screen "Home Screen" 1280x800, template "Template_Home"
   Circle "Circle_2" at 219,200 size 21x21
      Appearance <- "DATA_STATUS.LH_SWING_STATUS"
   SymbolLibrary "Symbol Library_1" at 1063,246 size 48x40
      Appearance <- "DATA_STATUS.IDFAN_STATUS"
   SymbolLibrary "Symbol Library_2" at 123,495 size 48x40
      Appearance <- "DATA_STATUS.LHFD_FAN_STATUS"
   SymbolLibrary "Symbol Library_3" at 123,276 size 48x40
      Appearance <- "DATA_STATUS.RHFD_FAN_STATUS"
   SymbolLibrary "Symbol Library_4" at 557,614 size 48x40
      Appearance <- "DATA_STATUS.FP1_STATUS"
   SymbolLibrary "Symbol Library_5" at 640,614 size 48x40
      Appearance <- "DATA_STATUS.FP2_STATUS"
   SymbolLibrary "Symbol Library_6" at 650,562 size 24x33
   SymbolLibrary "Symbol Library_7" at 570,562 size 24x33
   SymbolLibrary "Symbol Library_8" at 570,662 size 24x33
   SymbolLibrary "Symbol Library_9" at 650,662 size 24x33
   SymbolLibrary "Symbol Library_11" at 855,508 size 48x40
      Appearance <- "WORK_BIT.MPA_26"
   TextField "Text Field_8" at 212,700 size 136x22; Text 'from deaerator tank'
   IOField "IO Field_1" at 1037,346 size 97x30; FormatPattern 99.9
      ProcessValue <- "ANALOG_DISPLAY.ID_SPEED"
   TextField "Text Field_10" at 1101,350 size 21x22; Text 'Hz'
   IOField "IO Field_2" at 30,499 size 84x32; FormatPattern 99.9
      ProcessValue <- "ANALOG_DISPLAY.RHFD_SPEED"
   TextField "Text Field_11" at 90,504 size 21x22; Text 'Hz'
   IOField "IO Field_3" at 33,278 size 84x32; FormatPattern 99.9
      ProcessValue <- "ANALOG_DISPLAY.LHFD_SPEED"
   TextField "Text Field_12" at 94,283 size 21x22; Text 'Hz'
   Bar "Bar_1" at 348,299 size 288x126; MinimumValue 0; MaximumValue 100
      ProcessValue <- "ANALOG_DISPLAY.WATER_LEVEL"
   IOField "IO Field_4" at 356,160 size 97x30; FormatPattern 99.9
      ProcessValue <- "ANALOG_DISPLAY.STEAM_PRESSURE"
   TextField "Text Field_13" at 415,164 size 25x22; Text 'bar'
   IOField "IO Field_5" at 686,672 size 71x32; FormatPattern 99.9
      ProcessValue <- "ANALOG_DISPLAY.FP2_SPEED"
   TextField "Text Field_14" at 730,677 size 21x22; Text 'Hz'
   IOField "IO Field_6" at 472,671 size 83x32; FormatPattern 99.9
      ProcessValue <- "ANALOG_DISPLAY.FP1_SPEED"
   TextField "Text Field_15" at 533,676 size 21x22; Text 'Hz'
   IOField "IO Field_7" at 600,444 size 97x32; FormatPattern 99.9
      ProcessValue <- "ANALOG_DISPLAY.RHSTOKER_SPEED"
   IOField "IO Field_8" at 598,249 size 97x30; FormatPattern 99.9
      ProcessValue <- "ANALOG_DISPLAY.LHSTOKER_SPEED"
   TextField "Text Field_16" at 658,253 size 21x22; Text 'Hz'
   TextField "Text Field_17" at 658,449 size 21x22; Text 'Hz'
   Rectangle "Rectangle_5" at 256,196 size 11x23
      Appearance <- "DATA_STATUS.LH_SWING_STATUS"
   TextField "Text Field_18" at 224,203 size 10x14; Text 'M'
   Rectangle "Rectangle_6" at 256,388 size 13x22
      Appearance <- "DATA_STATUS.RH_SWING_STATUS"
   IOField "IO Field_9" at 442,541 size 97x32; FormatPattern 99.9
      ProcessValue <- "ANALOG_DISPLAY.PUMP_PRESSURE"
   TextField "Text Field_20" at 500,546 size 25x22; Text 'bar'
   IOField "IO Field_10" at 386,573 size 153x32; FormatPattern 99.9
      ProcessValue <- "ANALOG_DISPLAY.WATER_FLOWRATE"
   TextField "Text Field_21" at 491,578 size 43x22; Text 'm³/hr'
   IOField "IO Field_11" at 386,605 size 153x32; FormatPattern 999999.9
      ProcessValue <- "ANALOG_DISPLAY.TOTAL_WATER"
   TextField "Text Field_22" at 500,610 size 24x22; Text 'm³'
   IOField "IO Field_12" at 964,111 size 97x32; FormatPattern 99.9
      ProcessValue <- "ANALOG_DISPLAY.O2_LEVEL"
   TextField "Text Field_23" at 1029,116 size 19x22; Text '%'
   IOField "IO Field_13" at 964,143 size 97x32; FormatPattern 99.9
      ProcessValue <- "ANALOG_DISPLAY.CO2_LEVEL"
   TextField "Text Field_24" at 1029,148 size 19x22; Text '%'
   IOField "IO Field_14" at 964,175 size 121x30; FormatPattern 999.9
      ProcessValue <- "ANALOG_DISPLAY.FLUE_GAS_TEMP"
   TextField "Text Field_26" at 925,116 size 22x22; Text 'O²'
   TextField "Text Field_27" at 916,145 size 31x22; Text 'CO²'
   TextField "Text Field_28" at 868,176 size 80x22; Text 'FLUE TEMP'
   TextField "Text Field_29" at 1053,179 size 20x22; Text '°C'
   IOField "IO Field_15" at 173,108 size 153x29; FormatPattern 999999.9
      ProcessValue <- "ANALOG_DISPLAY.LH_TOTAL_COAL"
   TextField "Text Field_30" at 276,112 size 37x22; Text 'Tons'
   IOField "IO Field_16" at 171,299 size 153x29; FormatPattern 999999.9
      ProcessValue <- "ANALOG_DISPLAY.RH_TOTAL_COAL"
   TextField "Text Field_31" at 273,303 size 37x22; Text 'Tons'
   IOField "IO Field_17" at 259,650 size 108x32; FormatPattern 999.9
      ProcessValue <- "ANALOG_DISPLAY.WATER_TEMP"
   IOField "IO Field_18" at 123,422 size 121x30; FormatPattern 999.9
      ProcessValue <- "ANALOG_DISPLAY.RH_BURNBACK_TEMP"
   TextField "Text Field_34" at 199,422 size 10x10; Text 'Text'
   TextField "Text Field_35" at 211,426 size 20x22; Text '°C'
   IOField "IO Field_19" at 121,228 size 121x30; FormatPattern 999.9
      ProcessValue <- "ANALOG_DISPLAY.LH_BURNBACK_TEMP"
   TextField "Text Field_37" at 216,232 size 20x22; Text '°C'
   SymbolLibrary "Symbol Library_14" at 529,166 size 40x33
   GraphicView "Graphics View_23" at 706,181 size 40x22; Picture "3-D Gate valve"
   TextField "Text Field_38" at 368,449 size 83x22; Text 'RH STOKER'
   TextField "Text Field_39" at 358,258 size 81x22; Text 'LH STOKER'
   TextField "Text Field_40" at 1060,381 size 52x22; Text 'ID FAN'
   TextField "Text Field_41" at 37,313 size 76x22; Text 'LH FD FAN'
   TextField "Text Field_42" at 33,535 size 78x22; Text 'RH FD FAN'
   TextField "Text Field_46" at 168,332 size 64x22; Text 'RH COAL'
   TextField "Text Field_48" at 110,399 size 102x22; Text 'RH BURNBACK'
   TextField "Text Field_50" at 914,447 size 91x22; Text 'ASH VALVE 2'
   Circle "Circle_10" at 137,350 size 21x21
      Appearance <- "DATA_STATUS.RHFD_FAN_STATUS"
   TextField "Text Field_3" at 142,353 size 10x14; Text 'M'
   Circle "Circle_8" at 220,392 size 21x21
      Appearance <- "DATA_STATUS.RH_SWING_STATUS"
   TextField "Text Field_19" at 225,395 size 10x14; Text 'M'
   Circle "Circle_11" at 262,450 size 21x21
      Appearance <- "DATA_STATUS.RH_STOKER_STATUS"
   TextField "Text Field_5" at 267,453 size 10x14; Text 'M'
   Circle "Circle_3" at 573,450 size 21x21
      Appearance <- "DATA_STATUS.RH_STOKER_STATUS"
   Circle "Circle_4" at 137,571 size 21x21
      Appearance <- "DATA_STATUS.LHFD_FAN_STATUS"
   TextField "Text Field_1" at 142,574 size 10x14; Text 'M'
   Circle "Circle_7" at 1077,324 size 21x21
      Appearance <- "DATA_STATUS.IDFAN_STATUS"
   TextField "Text Field_7" at 1081,326 size 12x16; Text 'M'
   Circle "Circle_5" at 947,420 size 21x21
      Appearance <- "DATA_STATUS.RAV2_STATUS"
   TextField "Text Field_61" at 951,422 size 12x16; Text 'M'
   Circle "Circle_6" at 702,526 size 21x21
      Appearance <- "DATA_STATUS.RAV1_STATUS"
   TextField "Text Field_2" at 706,528 size 12x16; Text 'M'
   Button "Button_1" at 0,730 size 98x68; TextOff 'Text'; PictureOn "Home_1"; PictureOff "Home_1"
      on Click: ActivateScreen("Home Screen", 0)
   Button "Button_2" at 98,730 size 100x68; TextOn 'Pumps'; TextOff 'Pumps'
      on Click: ActivateScreen("Feed Pump", 0)
   Button "Button_3" at 198,730 size 90x68; TextOn 'Fans'; TextOff 'Fans'
      on Click: ActivateScreen("ID FD Fan", 0)
   Button "Button_4" at 288,730 size 100x68; TextOn 'Stoker'; TextOff 'Stoker'
      on Click: ActivateScreen("Stoker", 0)
   Button "Button_6" at 516,730 size 89x68; TextOff 'Setup'
      on Click: ActivateScreen("Setup", 0)
   Button "Button_11" at 1164,730 size 114x68; TextOff 'Trends'
      on Click: ActivateScreen("Trend Steam", 0)
   Button "Button_5" at 387,730 size 129x68; TextOff 'Coal Handling'
      on Click: ActivateScreen("Coal Handling", 0)
   Button "Button_7" at 604,730 size 210x68; TextOff 'Coal & Blowdown Setup'
      on Click: ActivateScreen("Coal Setup", 0)
   Button "Button_8" at 814,730 size 140x68; TextOff 'Front/Rear Undergrate'
      on Click: ActivateScreen("Front Undergrate Damper", 0)
   Button "Button_20" at 954,730 size 100x68; TextOff 'Alarm Setup'
      on Click: ActivateScreen("Alarm Setup", 0)
   Button "Button_21" at 1054,730 size 110x68; TextOff 'Alarm History'
      on Click: ActivateScreen("Alarm History", 0)
   TextField "Text Field_52" at 675,554 size 91x22; Text 'ASH VALVE 1'
   Circle "Circle_9" at 580,517 size 21x21
      Appearance <- "DATA_STATUS.ASH_CONV_STATUS"
   TextField "Text Field_43" at 584,519 size 12x16; Text 'M'
   TextField "Text Field_44" at 463,516 size 113x22; Text 'ASH CONVEYOR'
   TextField "Text Field_51" at 688,650 size 94x22; Text 'FEED PUMP 2'
   TextField "Text Field_53" at 461,649 size 94x22; Text 'FEED PUMP 1'
   TextField "Text Field_47" at 274,609 size 106x22; Text 'TOTAL WATER'
   TextField "Text Field_54" at 245,578 size 135x22; Text 'WATER FLOWRATE'
   TextField "Text Field_55" at 323,547 size 115x22; Text 'PUMP PRESSURE'
   TextField "Text Field_56" at 84,376 size 128x22; Text 'RH SWING CHUTE'
   TextField "Text Field_45" at 115,203 size 100x22; Text 'LH BURNBACK'
   TextField "Text Field_49" at 89,180 size 126x22; Text 'LH SWING CHUTE'
   TextField "Text Field_57" at 167,145 size 62x22; Text 'LH COAL'
   TextField "Text Field_58" at 358,134 size 124x22; Text 'STEAM PRESSURE'
   TextField "Text field_59" at 646,410 size 13x22; Text '0'
   TextField "Text field_60" at 642,388 size 21x22; Text '20'
   TextField "Text field_62" at 642,363 size 21x22; Text '40'
   TextField "Text field_63" at 642,338 size 21x22; Text '60'
   TextField "Text field_64" at 642,313 size 21x22; Text '80'
   TextField "Text field_65" at 638,288 size 29x22; Text '100'
   GraphicView "Graphic view_2" at 1184,120 size 66x412; Picture "Graphic_4"
   GraphicView "Graphic view_1" at 1178,513 size 80x14; Picture "Graphic_5"
   Button "Button_9" at 914,504 size 99x58; TextOff 'AUTOMATIC BLOWDOWN'
      on Click: function_efd93a16("Automatic Blowdown", 900, 370, -1, -1, 1)
   Circle "Circle_12" at 565,258 size 22x22
      Appearance <- "DATA_STATUS.LH_STOKER_STATUS"
   TextField "Text field_6" at 545,335 size 42x50; Text '%'
   IOField "IO Field_20" at 415,334 size 121x49; FormatPattern 999.9
      ProcessValue <- "ANALOG_DISPLAY.WATER_LEVEL"
   Circle "Circle_1" at 255,258 size 22x22
      Appearance <- "DATA_STATUS.LH_STOKER_STATUS"
   TextField "Text Field_4" at 261,262 size 10x14; Text 'M'
   TextField "Text Field_9" at 338,655 size 20x22; Text '°C'
   Button "Button_10" at 107,226 size 149x36; TextOff 'Text'
      on Click: function_efd93a16("BURN_BACK_OFFSET LH", 249, 122, -1, -1, 1)
   Button "Button_12" at 108,421 size 149x36; TextOff 'Text'
      on Click: function_efd93a16("BURN_BACK_OFFSET RH", 240, 436, -1, -1, 1)

screen "Alarm History" 1280x800, template "Template_All"
   TextField "Text Field_1" at 455,109 size 290x50; Text 'ALARM HISTORY'
   AlarmView "Alarm View_1" at 20,182 size 1244x536; ColumnTextDevice 'PLC'; ColumnTextAckGroup 'GR'; ColumnTextAlarmState 'Status'; ColumnTextAlarmText 'Text'; ColumnTextTime 'Time'; ColumnTextDate 'Date'; ColumnTextNumber 'No.'; AlarmLog "Alarm_History"
   Button "Button_1" at 0,730 size 98x68; TextOff 'Text'; PictureOn "Home_1"; PictureOff "Home_1"
      on Click: ActivateScreen("Home Screen", 0)
   Button "Button_2" at 98,730 size 100x68; TextOn 'Pumps'; TextOff 'Pumps'
      on Click: ActivateScreen("Feed Pump", 0)
   Button "Button_3" at 198,730 size 90x68; TextOn 'Fans'; TextOff 'Fans'
      on Click: ActivateScreen("ID FD Fan", 0)
   Button "Button_4" at 288,730 size 100x68; TextOn 'Stoker'; TextOff 'Stoker'
      on Click: ActivateScreen("Stoker", 0)
   Button "Button_6" at 516,730 size 89x68; TextOff 'Setup'
      on Click: ActivateScreen("Setup", 0)
   Button "Button_11" at 1164,730 size 114x68; TextOff 'Trends'
      on Click: ActivateScreen("Trend Steam", 0)
   Button "Button_18" at 387,730 size 129x68; TextOff 'Coal Handling'
      on Click: ActivateScreen("Coal Handling", 0)
   Button "Button_5" at 604,730 size 210x68; TextOff 'Coal & Blowdown Setup'
      on Click: ActivateScreen("Coal Setup", 0)
   Button "Button_19" at 814,730 size 140x68; TextOff 'Front/Rear Undergrate'
      on Click: ActivateScreen("Front Undergrate Damper", 0)
   Button "Button_20" at 954,730 size 100x68; TextOff 'Alarm Setup'
      on Click: ActivateScreen("Alarm Setup", 0)
   Button "Button_21" at 1054,730 size 110x68; TextOff 'Alarm History'
      on Click: ActivateScreen("Alarm History", 0)

screen "Feed Pump" 1280x800, template "Template_All"
   TextField "Text Field_1" at 515,108 size 221x50; Text 'FEED PUMPS'
   SymbolLibrary "Symbol Library_4" at 235,404 size 80x66
      Appearance <- "DATA_STATUS.FP1_STATUS"
   SymbolLibrary "Symbol Library_5" at 365,404 size 80x66
      Appearance <- "DATA_STATUS.FP2_STATUS"
   SymbolLibrary "Symbol Library_1" at 251,525 size 40x59
   SymbolLibrary "Symbol Library_2" at 387,525 size 40x59
   SymbolLibrary "Symbol Library_3" at 255,297 size 40x59
   SymbolLibrary "Symbol Library_8" at 387,297 size 40x59
   TextField "Text Field_2" at 43,614 size 146x22; Text 'From Deaerator Tank'
   Bar "Bar_1" at 616,253 size 208x373; MinimumValue 0; MaximumValue 100
      ProcessValue <- "ANALOG_DISPLAY.WATER_LEVEL"
   TextField "Text Field_3" at 636,219 size 143x37; Text 'Water Level'
   IOField "IO Field_12" at 632,632 size 172x41; FormatPattern 999.9
      ProcessValue <- "ANALOG_DISPLAY.WATER_LEVEL"
   TextField "Text Field_23" at 754,634 size 28x34; Text '%'
   IOField "IO Field_6" at 89,425 size 112x36; FormatPattern 99.9
      ProcessValue <- "ANALOG_DISPLAY.FP1_SPEED"
   TextField "Text Field_15" at 165,429 size 32x34; Text 'Hz'
   IOField "IO Field_7" at 475,425 size 112x36; FormatPattern 99.9
      ProcessValue <- "ANALOG_DISPLAY.FP2_SPEED"
   TextField "Text Field_16" at 547,429 size 32x34; Text 'Hz'
   Switch "Switch_1" at 910,268 size 240x79; TextOn 'AUTO'; CaptionText 'Switch'; TextOff 'HAND'
      ProcessValue <- "DATA_SWITCH.AUTO_FP"
      Appearance <- "DATA_SWITCH.AUTO_FP"
   Button "Button_8" at 910,349 size 240x79; TextOff 'SPEED UP'
      on Press: function_dd21b452("DATA_PARAMETER.HAND_REFF_FP", 2); function_b14e0dd5("PUMP_SPEED_UP", 0)
      Appearance <- "PUMP_SPEED_UP"
   Button "Button_9" at 910,430 size 240x79; TextOff 'SPEED DOWN'
      on Press: function_b9b71300("DATA_PARAMETER.HAND_REFF_FP", 2); function_b14e0dd5("PUMP_SPEED_DOWN", 0)
      Appearance <- "PUMP_SPEED_DOWN"
   IOField "IO Field_10" at 910,581 size 210x43; FormatPattern 99.9
      ProcessValue <- "ANALOG_DISPLAY.WATER_FLOWRATE"
   TextField "Text Field_21" at 1028,585 size 70x34; Text 'm³/hr'
   IOField "IO Field_11" at 245,668 size 192x39; FormatPattern 999999.9
      ProcessValue <- "ANALOG_DISPLAY.TOTAL_WATER"
   TextField "Text Field_22" at 386,669 size 37x34; Text 'm³'
   IOField "IO Field_9" at 289,206 size 110x38; FormatPattern 99.9
      ProcessValue <- "ANALOG_DISPLAY.PUMP_PRESSURE"
   TextField "Text Field_20" at 355,209 size 40x34; Text 'bar'
   TextField "Text Field_4" at 924,542 size 173x34; Text 'Water Flowrate'
   TextField "Text Field_5" at 253,167 size 194x37; Text 'Pumps Pressure'
   TextField "Text Field_6" at 73,356 size 160x70; Text 'Feed Pump 1 Speed'
   TextField "Text Field_7" at 453,356 size 160x70; Text 'Feed Pump 2 Speed'
   TextField "Text Field_9" at 267,630 size 143x37; Text 'Total Water'
   Button "Button_1" at 0,730 size 98x68; TextOff 'Text'; PictureOn "Home_1"; PictureOff "Home_1"
      on Click: ActivateScreen("Home Screen", 0)
   Button "Button_2" at 98,730 size 100x68; TextOn 'Pumps'; TextOff 'Pumps'
      on Click: ActivateScreen("Feed Pump", 0)
   Button "Button_3" at 198,730 size 90x68; TextOn 'Fans'; TextOff 'Fans'
      on Click: ActivateScreen("ID FD Fan", 0)
   Button "Button_4" at 288,730 size 100x68; TextOn 'Stoker'; TextOff 'Stoker'
      on Click: ActivateScreen("Stoker", 0)
   Button "Button_6" at 516,730 size 89x68; TextOff 'Setup'
      on Click: ActivateScreen("Setup", 0)
   Button "Button_11" at 1164,730 size 114x68; TextOff 'Trends'
      on Click: ActivateScreen("Trend Steam", 0)
   Button "Button_5" at 387,730 size 129x68; TextOff 'Coal Handling'
      on Click: ActivateScreen("Coal Handling", 0)
   Button "Button_7" at 605,730 size 210x68; TextOff 'Coal & Blowdown Setup'
      on Click: ActivateScreen("Coal Setup", 0)
   Button "Button_10" at 814,730 size 140x68; TextOff 'Front/Rear Undergrate'
      on Click: ActivateScreen("Front Undergrate Damper", 0)
   Button "Button_20" at 954,730 size 100x68; TextOff 'Alarm Setup'
      on Click: ActivateScreen("Alarm Setup", 0)
   Button "Button_21" at 1054,730 size 110x68; TextOff 'Alarm History'
      on Click: ActivateScreen("Alarm History", 0)

screen "Trend Steam" 1280x800, template "Template_All"
   Button "Button_1" at 4,735 size 182x64; TextOff 'Pumps'; PictureOff "Home_2"
      on Click: ActivateScreen("Home Screen", 0)
   Button "Button_2" at 550,735 size 182x64; TextOff 'Water Flow Trend'
      on Click: ActivateScreen("Trend Water Flow", 0)
   Button "Button_3" at 4,670 size 182x63; TextOff 'ID Fan Trend'
      on Click: ActivateScreen("Trend ID Fan", 0)
   Button "Button_4" at 732,735 size 182x64; TextOff 'Water Level Trend'
      on Click: ActivateScreen("Trend Water Level", 0)
   Button "Button_5" at 1096,735 size 182x64; TextOff 'Oxygen Level Trend'
      on Click: ActivateScreen("Trend O²", 0)
   Button "Button_6" at 914,735 size 182x64; TextOff 'Flue Temp Trend'
      on Click: ActivateScreen("Trend Flue Gas", 0)
   Button "Button_7" at 914,670 size 182x64; TextOff 'Water Temp Trend'
      on Click: ActivateScreen("Trend Water Temp", 0)
   TextField "Text Field_1" at 455,110 size 440x50; Text 'STEAM PRESSURE TREND'
   TrendView "Trend View_1" at 0,170 size 1280x490
   Button "Button_8" at 368,735 size 182x64; TextOff 'RH Stoker Trend'
      on Click: ActivateScreen("Trend RH Stoker", 0)
   Button "Button_9" at 186,735 size 182x64; TextOff 'LH Stoker Trend'
      on Click: ActivateScreen("Trend LH Stoker", 0)
   Button "Button_10" at 368,670 size 182x64; TextOff 'RH FD Fan Trend'
      on Click: ActivateScreen("Trend RH FD Fan", 0)
   Button "Button_11" at 186,670 size 182x64; TextOff 'LH FD Fan Trend'
      on Click: ActivateScreen("Trend LH FD Fan", 0)
   Button "Button_13" at 1096,670 size 182x64; TextOff 'CO² Level Trend'
      on Click: ActivateScreen("Trend CO²", 0)
   Button "Button_14" at 550,670 size 182x64; TextOff 'Feed Pump Speed Trend'
      on Click: ActivateScreen("Trend Pump Speed", 0)
   Button "Button_15" at 732,670 size 182x64; TextOff 'Pump Press Trend'
      on Click: ActivateScreen("Trend Pump Pressure", 0)

screen "Trend CO²" 1280x800, template "Template_All"
   TextField "Text Field_1" at 496,110 size 318x50; Text 'CO² LEVEL TREND'
   TrendView "Trend View_1" at 0,170 size 1280x490
   Button "Button_13" at 1096,670 size 182x64; TextOff 'Steam Press Trend'
      on Click: ActivateScreen("Trend Steam", 0)
   Button "Button_1" at 4,735 size 182x64; TextOff 'Pumps'; PictureOff "Home_2"
      on Click: ActivateScreen("Home Screen", 0)
   Button "Button_2" at 550,735 size 182x64; TextOff 'Water Flow Trend'
      on Click: ActivateScreen("Trend Water Flow", 0)
   Button "Button_3" at 4,670 size 182x63; TextOff 'ID Fan Trend'
      on Click: ActivateScreen("Trend ID Fan", 0)
   Button "Button_4" at 732,735 size 182x64; TextOff 'Water Level Trend'
      on Click: ActivateScreen("Trend Water Level", 0)
   Button "Button_5" at 1096,735 size 182x64; TextOff 'Oxygen Level Trend'
      on Click: ActivateScreen("Trend O²", 0)
   Button "Button_6" at 914,735 size 182x64; TextOff 'Flue Temp Trend'
      on Click: ActivateScreen("Trend Flue Gas", 0)
   Button "Button_7" at 914,670 size 182x64; TextOff 'Water Temp Trend'
      on Click: ActivateScreen("Trend Water Temp", 0)
   Button "Button_8" at 368,735 size 182x64; TextOff 'RH Stoker Trend'
      on Click: ActivateScreen("Trend RH Stoker", 0)
   Button "Button_9" at 186,735 size 182x64; TextOff 'LH Stoker Trend'
      on Click: ActivateScreen("Trend LH Stoker", 0)
   Button "Button_10" at 368,670 size 182x64; TextOff 'RH FD Fan Trend'
      on Click: ActivateScreen("Trend RH FD Fan", 0)
   Button "Button_11" at 186,670 size 182x64; TextOff 'LH FD Fan Trend'
      on Click: ActivateScreen("Trend LH FD Fan", 0)
   Button "Button_14" at 550,670 size 182x64; TextOff 'Feed Pump Speed Trend'
      on Click: ActivateScreen("Trend Pump Speed", 0)
   Button "Button_15" at 732,670 size 182x64; TextOff 'Pump Press Trend'
      on Click: ActivateScreen("Trend Pump Pressure", 0)

screen "Trend Flue Gas" 1280x800, template "Template_All"
   TextField "Text Field_1" at 481,112 size 405x50; Text 'FLUE GAS TEMP TREND'
   TrendView "Trend View_1" at 0,170 size 1280x490
   Button "Button_6" at 914,735 size 182x64; TextOff 'Steam Press Trend'
      on Click: ActivateScreen("Trend Steam", 0)
   Button "Button_1" at 4,735 size 182x64; TextOff 'Pumps'; PictureOff "Home_2"
      on Click: ActivateScreen("Home Screen", 0)
   Button "Button_2" at 550,735 size 182x64; TextOff 'Water Flow Trend'
      on Click: ActivateScreen("Trend Water Flow", 0)
   Button "Button_3" at 4,670 size 182x63; TextOff 'ID Fan Trend'
      on Click: ActivateScreen("Trend ID Fan", 0)
   Button "Button_4" at 732,735 size 182x64; TextOff 'Water Level Trend'
      on Click: ActivateScreen("Trend Water Level", 0)
   Button "Button_5" at 1096,735 size 182x64; TextOff 'Oxygen Level Trend'
      on Click: ActivateScreen("Trend O²", 0)
   Button "Button_8" at 914,670 size 182x64; TextOff 'Water Temp Trend'
      on Click: ActivateScreen("Trend Water Temp", 0)
   Button "Button_9" at 368,735 size 182x64; TextOff 'RH Stoker Trend'
      on Click: ActivateScreen("Trend RH Stoker", 0)
   Button "Button_10" at 186,735 size 182x64; TextOff 'LH Stoker Trend'
      on Click: ActivateScreen("Trend LH Stoker", 0)
   Button "Button_11" at 368,670 size 182x64; TextOff 'RH FD Fan Trend'
      on Click: ActivateScreen("Trend RH FD Fan", 0)
   Button "Button_12" at 186,670 size 182x64; TextOff 'LH FD Fan Trend'
      on Click: ActivateScreen("Trend LH FD Fan", 0)
   Button "Button_13" at 1096,670 size 182x64; TextOff 'CO² Level Trend'
      on Click: ActivateScreen("Trend CO²", 0)
   Button "Button_14" at 550,670 size 182x64; TextOff 'Feed Pump Speed Trend'
      on Click: ActivateScreen("Trend Pump Speed", 0)
   Button "Button_15" at 732,670 size 182x64; TextOff 'Pump Press Trend'
      on Click: ActivateScreen("Trend Pump Pressure", 0)

screen "Trend ID Fan" 1280x800, template "Template_All"
   TrendView "Trend View_1" at 0,170 size 1280x490
   TextField "Text Field_1" at 482,113 size 376x50; Text 'ID FAN SPEED TREND'
   Button "Button_3" at 4,670 size 182x64; TextOff 'Steam Press Trend'
      on Click: ActivateScreen("Trend Steam", 0)
   Button "Button_1" at 4,735 size 182x64; TextOff 'Pumps'; PictureOff "Home_2"
      on Click: ActivateScreen("Home Screen", 0)
   Button "Button_2" at 550,735 size 182x64; TextOff 'Water Flow Trend'
      on Click: ActivateScreen("Trend Water Flow", 0)
   Button "Button_5" at 732,735 size 182x64; TextOff 'Water Level Trend'
      on Click: ActivateScreen("Trend Water Level", 0)
   Button "Button_6" at 1096,735 size 182x64; TextOff 'Oxygen Level Trend'
      on Click: ActivateScreen("Trend O²", 0)
   Button "Button_7" at 914,735 size 182x64; TextOff 'Flue Temp Trend'
      on Click: ActivateScreen("Trend Flue Gas", 0)
   Button "Button_8" at 914,670 size 182x64; TextOff 'Water Temp Trend'
      on Click: ActivateScreen("Trend Water Temp", 0)
   Button "Button_9" at 368,735 size 182x64; TextOff 'RH Stoker Trend'
      on Click: ActivateScreen("Trend RH Stoker", 0)
   Button "Button_10" at 186,735 size 182x64; TextOff 'LH Stoker Trend'
      on Click: ActivateScreen("Trend LH Stoker", 0)
   Button "Button_11" at 368,670 size 182x64; TextOff 'RH FD Fan Trend'
      on Click: ActivateScreen("Trend RH FD Fan", 0)
   Button "Button_12" at 186,670 size 182x64; TextOff 'LH FD Fan Trend'
      on Click: ActivateScreen("Trend LH FD Fan", 0)
   Button "Button_13" at 1096,670 size 182x64; TextOff 'CO² Level Trend'
      on Click: ActivateScreen("Trend CO²", 0)
   Button "Button_14" at 550,670 size 182x64; TextOff 'Feed Pump Speed Trend'
      on Click: ActivateScreen("Trend Pump Speed", 0)
   Button "Button_15" at 732,670 size 182x64; TextOff 'Pump Press Trend'
      on Click: ActivateScreen("Trend Pump Pressure", 0)

screen "Trend LH Stoker" 1280x800, template "Template_All"
   TrendView "Trend View_1" at 0,170 size 1280x490
   Button "Button_9" at 186,735 size 182x64; TextOff 'Steam Press Trend'
      on Click: ActivateScreen("Trend Steam", 0)
   Button "Button_1" at 4,735 size 182x64; TextOff 'Pumps'; PictureOff "Home_2"
      on Click: ActivateScreen("Home Screen", 0)
   Button "Button_2" at 550,735 size 182x64; TextOff 'Water Flow Trend'
      on Click: ActivateScreen("Trend Water Flow", 0)
   Button "Button_3" at 4,670 size 182x63; TextOff 'ID Fan Trend'
      on Click: ActivateScreen("Trend ID Fan", 0)
   Button "Button_4" at 732,735 size 182x64; TextOff 'Water Level Trend'
      on Click: ActivateScreen("Trend Water Level", 0)
   Button "Button_5" at 1096,735 size 182x64; TextOff 'Oxygen Level Trend'
      on Click: ActivateScreen("Trend O²", 0)
   Button "Button_6" at 914,735 size 182x64; TextOff 'Flue Temp Trend'
      on Click: ActivateScreen("Trend Flue Gas", 0)
   Button "Button_7" at 914,670 size 182x64; TextOff 'Water Temp Trend'
      on Click: ActivateScreen("Trend Water Temp", 0)
   Button "Button_8" at 368,735 size 182x64; TextOff 'RH Stoker Trend'
      on Click: ActivateScreen("Trend RH Stoker", 0)
   Button "Button_11" at 368,670 size 182x64; TextOff 'RH FD Fan Trend'
      on Click: ActivateScreen("Trend RH FD Fan", 0)
   Button "Button_12" at 186,670 size 182x64; TextOff 'LH FD Fan Trend'
      on Click: ActivateScreen("Trend LH FD Fan", 0)
   Button "Button_13" at 1096,670 size 182x64; TextOff 'CO² Level Trend'
      on Click: ActivateScreen("Trend CO²", 0)
   Button "Button_14" at 550,670 size 182x64; TextOff 'Feed Pump Speed Trend'
      on Click: ActivateScreen("Trend Pump Speed", 0)
   Button "Button_15" at 732,670 size 182x64; TextOff 'Pump Press Trend'
      on Click: ActivateScreen("Trend Pump Pressure", 0)
   TextField "Text Field_1" at 465,113 size 450x50; Text 'LH STOKER SPEED TREND'

screen "Trend LH FD Fan" 1280x800, template "Template_All"
   TextField "Text Field_1" at 444,113 size 439x50; Text 'LH FD FAN SPEED TREND'
   TrendView "Trend View_1" at 0,170 size 1280x490
   Button "Button_11" at 186,670 size 182x64; TextOff 'Steam Press Trend'
      on Click: ActivateScreen("Trend Steam", 0)
   Button "Button_1" at 4,735 size 182x64; TextOff 'Pumps'; PictureOff "Home_2"
      on Click: ActivateScreen("Home Screen", 0)
   Button "Button_2" at 550,735 size 182x64; TextOff 'Water Flow Trend'
      on Click: ActivateScreen("Trend Water Flow", 0)
   Button "Button_3" at 4,670 size 182x63; TextOff 'ID Fan Trend'
      on Click: ActivateScreen("Trend ID Fan", 0)
   Button "Button_4" at 732,735 size 182x64; TextOff 'Water Level Trend'
      on Click: ActivateScreen("Trend Water Level", 0)
   Button "Button_5" at 1096,735 size 182x64; TextOff 'Oxygen Level Trend'
      on Click: ActivateScreen("Trend O²", 0)
   Button "Button_6" at 914,735 size 182x64; TextOff 'Flue Temp Trend'
      on Click: ActivateScreen("Trend Flue Gas", 0)
   Button "Button_7" at 914,670 size 182x64; TextOff 'Water Temp Trend'
      on Click: ActivateScreen("Trend Water Temp", 0)
   Button "Button_8" at 368,735 size 182x64; TextOff 'RH Stoker Trend'
      on Click: ActivateScreen("Trend RH Stoker", 0)
   Button "Button_9" at 186,735 size 182x64; TextOff 'LH Stoker Trend'
      on Click: ActivateScreen("Trend LH Stoker", 0)
   Button "Button_10" at 368,670 size 182x64; TextOff 'RH FD Fan Trend'
      on Click: ActivateScreen("Trend RH FD Fan", 0)
   Button "Button_13" at 1096,670 size 182x64; TextOff 'CO² Level Trend'
      on Click: ActivateScreen("Trend CO²", 0)
   Button "Button_14" at 550,670 size 182x64; TextOff 'Feed Pump Speed Trend'
      on Click: ActivateScreen("Trend Pump Speed", 0)
   Button "Button_15" at 732,670 size 182x64; TextOff 'Pump Press Trend'
      on Click: ActivateScreen("Trend Pump Pressure", 0)

screen "Trend O²" 1280x800, template "Template_All"
   TextField "Text Field_1" at 468,111 size 391x50; Text 'OXYGEN LEVEL TREND'
   TrendView "Trend View_1" at 0,170 size 1280x490
   Button "Button_5" at 1096,735 size 182x64; TextOff 'Steam Press Trend'
      on Click: ActivateScreen("Trend Steam", 0)
   Button "Button_1" at 4,735 size 182x64; TextOff 'Pumps'; PictureOff "Home_2"
      on Click: ActivateScreen("Home Screen", 0)
   Button "Button_2" at 550,735 size 182x64; TextOff 'Water Flow Trend'
      on Click: ActivateScreen("Trend Water Flow", 0)
   Button "Button_3" at 4,670 size 182x63; TextOff 'ID Fan Trend'
      on Click: ActivateScreen("Trend ID Fan", 0)
   Button "Button_4" at 732,735 size 182x64; TextOff 'Water Level Trend'
      on Click: ActivateScreen("Trend Water Level", 0)
   Button "Button_7" at 914,735 size 182x64; TextOff 'Flue Temp Trend'
      on Click: ActivateScreen("Trend Flue Gas", 0)
   Button "Button_8" at 914,670 size 182x64; TextOff 'Water Temp Trend'
      on Click: ActivateScreen("Trend Water Temp", 0)
   Button "Button_9" at 368,735 size 182x64; TextOff 'RH Stoker Trend'
      on Click: ActivateScreen("Trend RH Stoker", 0)
   Button "Button_10" at 186,735 size 182x64; TextOff 'LH Stoker Trend'
      on Click: ActivateScreen("Trend LH Stoker", 0)
   Button "Button_11" at 368,670 size 182x64; TextOff 'RH FD Fan Trend'
      on Click: ActivateScreen("Trend RH FD Fan", 0)
   Button "Button_12" at 186,670 size 182x64; TextOff 'LH FD Fan Trend'
      on Click: ActivateScreen("Trend LH FD Fan", 0)
   Button "Button_13" at 1096,670 size 182x64; TextOff 'CO² Level Trend'
      on Click: ActivateScreen("Trend CO²", 0)
   Button "Button_14" at 550,670 size 182x64; TextOff 'Feed Pump Speed Trend'
      on Click: ActivateScreen("Trend Pump Speed", 0)
   Button "Button_15" at 732,670 size 182x64; TextOff 'Pump Press Trend'
      on Click: ActivateScreen("Trend Pump Pressure", 0)

screen "Trend Pump Pressure" 1280x800, template "Template_All"
   TextField "Text Field_1" at 456,112 size 441x50; Text 'PUMPS PRESSURE TREND'
   TrendView "Trend View_1" at 0,170 size 1280x490
   Button "Button_15" at 732,670 size 182x64; TextOff 'Steam Press Trend'
      on Click: ActivateScreen("Trend Steam", 0)
   Button "Button_1" at 4,735 size 182x64; TextOff 'Pumps'; PictureOff "Home_2"
      on Click: ActivateScreen("Home Screen", 0)
   Button "Button_2" at 550,735 size 182x64; TextOff 'Water Flow Trend'
      on Click: ActivateScreen("Trend Water Flow", 0)
   Button "Button_3" at 4,670 size 182x63; TextOff 'ID Fan Trend'
      on Click: ActivateScreen("Trend ID Fan", 0)
   Button "Button_4" at 732,735 size 182x64; TextOff 'Water Level Trend'
      on Click: ActivateScreen("Trend Water Level", 0)
   Button "Button_5" at 1096,735 size 182x64; TextOff 'Oxygen Level Trend'
      on Click: ActivateScreen("Trend O²", 0)
   Button "Button_6" at 914,735 size 182x64; TextOff 'Flue Temp Trend'
      on Click: ActivateScreen("Trend Flue Gas", 0)
   Button "Button_7" at 914,670 size 182x64; TextOff 'Water Temp Trend'
      on Click: ActivateScreen("Trend Water Temp", 0)
   Button "Button_8" at 368,735 size 182x64; TextOff 'RH Stoker Trend'
      on Click: ActivateScreen("Trend RH Stoker", 0)
   Button "Button_9" at 186,735 size 182x64; TextOff 'LH Stoker Trend'
      on Click: ActivateScreen("Trend LH Stoker", 0)
   Button "Button_10" at 368,670 size 182x64; TextOff 'RH FD Fan Trend'
      on Click: ActivateScreen("Trend RH FD Fan", 0)
   Button "Button_11" at 186,670 size 182x64; TextOff 'LH FD Fan Trend'
      on Click: ActivateScreen("Trend LH FD Fan", 0)
   Button "Button_13" at 1096,670 size 182x64; TextOff 'CO² Level Trend'
      on Click: ActivateScreen("Trend CO²", 0)
   Button "Button_14" at 550,670 size 182x64; TextOff 'Feed Pump Speed Trend'
      on Click: ActivateScreen("Trend Pump Speed", 0)

screen "Trend Pump Speed" 1280x800, template "Template_All"
   TrendView "Trend View_1" at 0,170 size 1280x490
   TextField "Text Field_1" at 435,112 size 473x50; Text 'FEED PUMPS SPEED TREND'
   Button "Button_14" at 550,670 size 182x64; TextOff 'Steam Press Trend'
      on Click: ActivateScreen("Trend Steam", 0)
   Button "Button_1" at 4,735 size 182x64; TextOff 'Pumps'; PictureOff "Home_2"
      on Click: ActivateScreen("Home Screen", 0)
   Button "Button_2" at 550,735 size 182x64; TextOff 'Water Flow Trend'
      on Click: ActivateScreen("Trend Water Flow", 0)
   Button "Button_3" at 4,670 size 182x63; TextOff 'ID Fan Trend'
      on Click: ActivateScreen("Trend ID Fan", 0)
   Button "Button_4" at 732,735 size 182x64; TextOff 'Water Level Trend'
      on Click: ActivateScreen("Trend Water Level", 0)
   Button "Button_5" at 1096,735 size 182x64; TextOff 'Oxygen Level Trend'
      on Click: ActivateScreen("Trend O²", 0)
   Button "Button_6" at 914,735 size 182x64; TextOff 'Flue Temp Trend'
      on Click: ActivateScreen("Trend Flue Gas", 0)
   Button "Button_7" at 914,670 size 182x64; TextOff 'Water Temp Trend'
      on Click: ActivateScreen("Trend Water Temp", 0)
   Button "Button_8" at 368,735 size 182x64; TextOff 'RH Stoker Trend'
      on Click: ActivateScreen("Trend RH Stoker", 0)
   Button "Button_9" at 186,735 size 182x64; TextOff 'LH Stoker Trend'
      on Click: ActivateScreen("Trend LH Stoker", 0)
   Button "Button_10" at 368,670 size 182x64; TextOff 'RH FD Fan Trend'
      on Click: ActivateScreen("Trend RH FD Fan", 0)
   Button "Button_11" at 186,670 size 182x64; TextOff 'LH FD Fan Trend'
      on Click: ActivateScreen("Trend LH FD Fan", 0)
   Button "Button_13" at 1096,670 size 182x64; TextOff 'CO² Level Trend'
      on Click: ActivateScreen("Trend CO²", 0)
   Button "Button_15" at 732,670 size 182x64; TextOff 'Pump Press Trend'
      on Click: ActivateScreen("Trend Pump Pressure", 0)

screen "Trend RH Stoker" 1280x800, template "Template_All"
   TextField "Text Field_1" at 465,113 size 455x50; Text 'RH STOKER SPEED TREND'
   TrendView "Trend View_1" at 0,170 size 1280x490
   Button "Button_8" at 368,735 size 182x64; TextOff 'Steam Press Trend'
      on Click: ActivateScreen("Trend Steam", 0)
   Button "Button_1" at 4,735 size 182x64; TextOff 'Pumps'; PictureOff "Home_2"
      on Click: ActivateScreen("Home Screen", 0)
   Button "Button_2" at 550,735 size 182x64; TextOff 'Water Flow Trend'
      on Click: ActivateScreen("Trend Water Flow", 0)
   Button "Button_3" at 4,670 size 182x63; TextOff 'ID Fan Trend'
      on Click: ActivateScreen("Trend ID Fan", 0)
   Button "Button_4" at 732,735 size 182x64; TextOff 'Water Level Trend'
      on Click: ActivateScreen("Trend Water Level", 0)
   Button "Button_5" at 1096,735 size 182x64; TextOff 'Oxygen Level Trend'
      on Click: ActivateScreen("Trend O²", 0)
   Button "Button_6" at 914,735 size 182x64; TextOff 'Flue Temp Trend'
      on Click: ActivateScreen("Trend Flue Gas", 0)
   Button "Button_7" at 914,670 size 182x64; TextOff 'Water Temp Trend'
      on Click: ActivateScreen("Trend Water Temp", 0)
   Button "Button_10" at 186,735 size 182x64; TextOff 'LH Stoker Trend'
      on Click: ActivateScreen("Trend LH Stoker", 0)
   Button "Button_11" at 368,670 size 182x64; TextOff 'RH FD Fan Trend'
      on Click: ActivateScreen("Trend RH FD Fan", 0)
   Button "Button_12" at 186,670 size 182x64; TextOff 'LH FD Fan Trend'
      on Click: ActivateScreen("Trend LH FD Fan", 0)
   Button "Button_13" at 1096,670 size 182x64; TextOff 'CO² Level Trend'
      on Click: ActivateScreen("Trend CO²", 0)
   Button "Button_14" at 550,670 size 182x64; TextOff 'Feed Pump Speed Trend'
      on Click: ActivateScreen("Trend Pump Speed", 0)
   Button "Button_15" at 732,670 size 182x64; TextOff 'Pump Press Trend'
      on Click: ActivateScreen("Trend Pump Pressure", 0)

screen "Trend RH FD Fan" 1280x800, template "Template_All"
   TextField "Text Field_1" at 434,113 size 444x50; Text 'RH FD FAN SPEED TREND'
   TrendView "Trend View_1" at 0,170 size 1280x490
   Button "Button_10" at 368,670 size 182x64; TextOff 'Steam Press Trend'
      on Click: ActivateScreen("Trend Steam", 0)
   Button "Button_1" at 4,735 size 182x64; TextOff 'Pumps'; PictureOff "Home_2"
      on Click: ActivateScreen("Home Screen", 0)
   Button "Button_2" at 550,735 size 182x64; TextOff 'Water Flow Trend'
      on Click: ActivateScreen("Trend Water Flow", 0)
   Button "Button_3" at 4,670 size 182x63; TextOff 'ID Fan Trend'
      on Click: ActivateScreen("Trend ID Fan", 0)
   Button "Button_4" at 732,735 size 182x64; TextOff 'Water Level Trend'
      on Click: ActivateScreen("Trend Water Level", 0)
   Button "Button_5" at 1096,735 size 182x64; TextOff 'Oxygen Level Trend'
      on Click: ActivateScreen("Trend O²", 0)
   Button "Button_6" at 914,735 size 182x64; TextOff 'Flue Temp Trend'
      on Click: ActivateScreen("Trend Flue Gas", 0)
   Button "Button_7" at 914,670 size 182x64; TextOff 'Water Temp Trend'
      on Click: ActivateScreen("Trend Water Temp", 0)
   Button "Button_8" at 368,735 size 182x64; TextOff 'RH Stoker Trend'
      on Click: ActivateScreen("Trend RH Stoker", 0)
   Button "Button_9" at 186,735 size 182x64; TextOff 'LH Stoker Trend'
      on Click: ActivateScreen("Trend LH Stoker", 0)
   Button "Button_12" at 186,670 size 182x64; TextOff 'LH FD Fan Trend'
      on Click: ActivateScreen("Trend LH FD Fan", 0)
   Button "Button_13" at 1096,670 size 182x64; TextOff 'CO² Level Trend'
      on Click: ActivateScreen("Trend CO²", 0)
   Button "Button_14" at 550,670 size 182x64; TextOff 'Feed Pump Speed Trend'
      on Click: ActivateScreen("Trend Pump Speed", 0)
   Button "Button_15" at 732,670 size 182x64; TextOff 'Pump Press Trend'
      on Click: ActivateScreen("Trend Pump Pressure", 0)

screen "Trend Water Flow" 1280x800, template "Template_All"
   TrendView "Trend View_1" at 0,170 size 1280x490
   TextField "Text Field_1" at 494,111 size 370x50; Text 'WATER FLOW TREND'
   Button "Button_2" at 550,735 size 182x64; TextOff 'Steam Press Trend'
      on Click: ActivateScreen("Trend Steam", 0)
   Button "Button_1" at 4,735 size 182x64; TextOff 'Pumps'; PictureOff "Home_2"
      on Click: ActivateScreen("Home Screen", 0)
   Button "Button_4" at 4,670 size 182x63; TextOff 'ID Fan Trend'
      on Click: ActivateScreen("Trend ID Fan", 0)
   Button "Button_5" at 732,735 size 182x64; TextOff 'Water Level Trend'
      on Click: ActivateScreen("Trend Water Level", 0)
   Button "Button_6" at 1096,735 size 182x64; TextOff 'Oxygen Level Trend'
      on Click: ActivateScreen("Trend O²", 0)
   Button "Button_7" at 914,735 size 182x64; TextOff 'Flue Temp Trend'
      on Click: ActivateScreen("Trend Flue Gas", 0)
   Button "Button_8" at 914,670 size 182x64; TextOff 'Water Temp Trend'
      on Click: ActivateScreen("Trend Water Temp", 0)
   Button "Button_9" at 368,735 size 182x64; TextOff 'RH Stoker Trend'
      on Click: ActivateScreen("Trend RH Stoker", 0)
   Button "Button_10" at 186,735 size 182x64; TextOff 'LH Stoker Trend'
      on Click: ActivateScreen("Trend LH Stoker", 0)
   Button "Button_11" at 368,670 size 182x64; TextOff 'RH FD Fan Trend'
      on Click: ActivateScreen("Trend RH FD Fan", 0)
   Button "Button_12" at 186,670 size 182x64; TextOff 'LH FD Fan Trend'
      on Click: ActivateScreen("Trend LH FD Fan", 0)
   Button "Button_13" at 1096,670 size 182x64; TextOff 'CO² Level Trend'
      on Click: ActivateScreen("Trend CO²", 0)
   Button "Button_14" at 550,670 size 182x64; TextOff 'Feed Pump Speed Trend'
      on Click: ActivateScreen("Trend Pump Speed", 0)
   Button "Button_15" at 732,670 size 182x64; TextOff 'Pump Press Trend'
      on Click: ActivateScreen("Trend Pump Pressure", 0)

screen "Trend Water Level" 1280x800, template "Template_All"
   TextField "Text Field_1" at 481,111 size 373x50; Text 'WATER LEVEL TREND'
   TrendView "Trend View_1" at 0,170 size 1280x490
   Button "Button_4" at 732,735 size 182x64; TextOff 'Steam Press Trend'
      on Click: ActivateScreen("Trend Steam", 0)
   Button "Button_1" at 4,735 size 182x64; TextOff 'Pumps'; PictureOff "Home_2"
      on Click: ActivateScreen("Home Screen", 0)
   Button "Button_2" at 550,735 size 182x64; TextOff 'Water Flow Trend'
      on Click: ActivateScreen("Trend Water Flow", 0)
   Button "Button_3" at 4,670 size 182x63; TextOff 'ID Fan Trend'
      on Click: ActivateScreen("Trend ID Fan", 0)
   Button "Button_6" at 1096,735 size 182x64; TextOff 'Oxygen Level Trend'
      on Click: ActivateScreen("Trend O²", 0)
   Button "Button_7" at 914,735 size 182x64; TextOff 'Flue Temp Trend'
      on Click: ActivateScreen("Trend Flue Gas", 0)
   Button "Button_8" at 914,670 size 182x64; TextOff 'Water Temp Trend'
      on Click: ActivateScreen("Trend Water Temp", 0)
   Button "Button_9" at 368,735 size 182x64; TextOff 'RH Stoker Trend'
      on Click: ActivateScreen("Trend RH Stoker", 0)
   Button "Button_10" at 186,735 size 182x64; TextOff 'LH Stoker Trend'
      on Click: ActivateScreen("Trend LH Stoker", 0)
   Button "Button_11" at 368,670 size 182x64; TextOff 'RH FD Fan Trend'
      on Click: ActivateScreen("Trend RH FD Fan", 0)
   Button "Button_12" at 186,670 size 182x64; TextOff 'LH FD Fan Trend'
      on Click: ActivateScreen("Trend LH FD Fan", 0)
   Button "Button_13" at 1096,670 size 182x64; TextOff 'CO² Level Trend'
      on Click: ActivateScreen("Trend CO²", 0)
   Button "Button_14" at 550,670 size 182x64; TextOff 'Feed Pump Speed Trend'
      on Click: ActivateScreen("Trend Pump Speed", 0)
   Button "Button_15" at 732,670 size 182x64; TextOff 'Pump Press Trend'
      on Click: ActivateScreen("Trend Pump Pressure", 0)

screen "Trend Water Temp" 1280x800, template "Template_All"
   TextField "Text Field_1" at 481,113 size 363x50; Text 'WATER TEMP TREND'
   TrendView "Trend View_1" at 0,170 size 1280x490
   Button "Button_7" at 914,670 size 182x64; TextOff 'Steam Press Trend'
      on Click: ActivateScreen("Trend Steam", 0)
   Button "Button_1" at 4,735 size 182x64; TextOff 'Pumps'; PictureOff "Home_2"
      on Click: ActivateScreen("Home Screen", 0)
   Button "Button_2" at 550,735 size 182x64; TextOff 'Water Flow Trend'
      on Click: ActivateScreen("Trend Water Flow", 0)
   Button "Button_3" at 4,670 size 182x63; TextOff 'ID Fan Trend'
      on Click: ActivateScreen("Trend ID Fan", 0)
   Button "Button_4" at 732,735 size 182x64; TextOff 'Water Level Trend'
      on Click: ActivateScreen("Trend Water Level", 0)
   Button "Button_5" at 1096,735 size 182x64; TextOff 'Oxygen Level Trend'
      on Click: ActivateScreen("Trend O²", 0)
   Button "Button_6" at 914,735 size 182x64; TextOff 'Flue Temp Trend'
      on Click: ActivateScreen("Trend Flue Gas", 0)
   Button "Button_9" at 368,735 size 182x64; TextOff 'RH Stoker Trend'
      on Click: ActivateScreen("Trend RH Stoker", 0)
   Button "Button_10" at 186,735 size 182x64; TextOff 'LH Stoker Trend'
      on Click: ActivateScreen("Trend LH Stoker", 0)
   Button "Button_11" at 368,670 size 182x64; TextOff 'RH FD Fan Trend'
      on Click: ActivateScreen("Trend RH FD Fan", 0)
   Button "Button_12" at 186,670 size 182x64; TextOff 'LH FD Fan Trend'
      on Click: ActivateScreen("Trend LH FD Fan", 0)
   Button "Button_13" at 1096,670 size 182x64; TextOff 'CO² Level Trend'
      on Click: ActivateScreen("Trend CO²", 0)
   Button "Button_14" at 550,670 size 182x64; TextOff 'Feed Pump Speed Trend'
      on Click: ActivateScreen("Trend Pump Speed", 0)
   Button "Button_15" at 732,670 size 182x64; TextOff 'Pump Press Trend'
      on Click: ActivateScreen("Trend Pump Pressure", 0)

screen "Trend PID FD Fan" 1280x800, template "Template_All"
   TrendView "Trend View_1" at 50,174 size 1186x542
   TextField "Text field_1" at 541,111 size 204x50; Text 'PID FD FAN'
   Button "Button_1" at 0,730 size 98x68; TextOff 'Text'; PictureOn "Home_1"; PictureOff "Home_1"
      on Click: ActivateScreen("Home Screen", 0)
   Button "Button_2" at 98,730 size 100x68; TextOn 'Pumps'; TextOff 'Pumps'
      on Click: ActivateScreen("Feed Pump", 0)
   Button "Button_3" at 198,730 size 90x68; TextOn 'Fans'; TextOff 'Fans'
      on Click: ActivateScreen("ID FD Fan", 0)
   Button "Button_4" at 288,730 size 100x68; TextOn 'Stoker'; TextOff 'Stoker'
      on Click: ActivateScreen("Stoker", 0)
   Button "Button_6" at 516,730 size 89x68; TextOff 'Setup'
      on Click: ActivateScreen("Setup", 0)
   Button "Button_11" at 1164,730 size 114x68; TextOff 'Trends'
      on Click: ActivateScreen("Trend Steam", 0)
   Button "Button_5" at 387,730 size 129x68; TextOff 'Coal Handling'
      on Click: ActivateScreen("Coal Handling", 0)
   Button "Button_7" at 604,730 size 210x68; TextOff 'Coal & Blowdown Setup'
      on Click: ActivateScreen("Coal Setup", 0)
   Button "Button_8" at 814,730 size 140x68; TextOff 'Front/Rear Undergrate'
      on Click: ActivateScreen("Front Undergrate Damper", 0)
   Button "Button_20" at 954,730 size 100x68; TextOff 'Alarm Setup'
      on Click: ActivateScreen("Alarm Setup", 0)
   Button "Button_21" at 1054,730 size 110x68; TextOff 'Alarm History'
      on Click: ActivateScreen("Alarm History", 0)

screen "Trend PID Pump" 1280x800, template "Template_All"
   TrendView "Trend View_1" at 44,174 size 1186x542
   TextField "Text field_1" at 561,113 size 174x50; Text 'PID PUMP'
   Button "Button_1" at 0,730 size 98x68; TextOff 'Text'; PictureOn "Home_1"; PictureOff "Home_1"
      on Click: ActivateScreen("Home Screen", 0)
   Button "Button_2" at 98,730 size 100x68; TextOn 'Pumps'; TextOff 'Pumps'
      on Click: ActivateScreen("Feed Pump", 0)
   Button "Button_3" at 198,730 size 90x68; TextOn 'Fans'; TextOff 'Fans'
      on Click: ActivateScreen("ID FD Fan", 0)
   Button "Button_4" at 288,730 size 100x68; TextOn 'Stoker'; TextOff 'Stoker'
      on Click: ActivateScreen("Stoker", 0)
   Button "Button_6" at 516,730 size 89x68; TextOff 'Setup'
      on Click: ActivateScreen("Setup", 0)
   Button "Button_11" at 1164,730 size 114x68; TextOff 'Trends'
      on Click: ActivateScreen("Trend Steam", 0)
   Button "Button_5" at 387,730 size 129x68; TextOff 'Coal Handling'
      on Click: ActivateScreen("Coal Handling", 0)
   Button "Button_7" at 604,730 size 210x68; TextOff 'Coal & Blowdown Setup'
      on Click: ActivateScreen("Coal Setup", 0)
   Button "Button_8" at 814,730 size 140x68; TextOff 'Front/Rear Undergrate'
      on Click: ActivateScreen("Front Undergrate Damper", 0)
   Button "Button_20" at 954,730 size 100x68; TextOff 'Alarm Setup'
      on Click: ActivateScreen("Alarm Setup", 0)
   Button "Button_21" at 1054,730 size 110x68; TextOff 'Alarm History'
      on Click: ActivateScreen("Alarm History", 0)

screen "Trend PID Stoker" 1280x800, template "Template_All"
   TrendView "Trend View_1" at 44,174 size 1186x542
   TextField "Text field_1" at 544,111 size 215x50; Text 'PID STOKER'
   Button "Button_1" at 0,730 size 98x68; TextOff 'Text'; PictureOn "Home_1"; PictureOff "Home_1"
      on Click: ActivateScreen("Home Screen", 0)
   Button "Button_2" at 98,730 size 100x68; TextOn 'Pumps'; TextOff 'Pumps'
      on Click: ActivateScreen("Feed Pump", 0)
   Button "Button_3" at 198,730 size 90x68; TextOn 'Fans'; TextOff 'Fans'
      on Click: ActivateScreen("ID FD Fan", 0)
   Button "Button_4" at 288,730 size 100x68; TextOn 'Stoker'; TextOff 'Stoker'
      on Click: ActivateScreen("Stoker", 0)
   Button "Button_6" at 516,730 size 89x68; TextOff 'Setup'
      on Click: ActivateScreen("Setup", 0)
   Button "Button_11" at 1164,730 size 114x68; TextOff 'Trends'
      on Click: ActivateScreen("Trend Steam", 0)
   Button "Button_5" at 387,730 size 129x68; TextOff 'Coal Handling'
      on Click: ActivateScreen("Coal Handling", 0)
   Button "Button_7" at 604,730 size 210x68; TextOff 'Coal & Blowdown Setup'
      on Click: ActivateScreen("Coal Setup", 0)
   Button "Button_8" at 814,730 size 140x68; TextOff 'Front/Rear Undergrate'
      on Click: ActivateScreen("Front Undergrate Damper", 0)
   Button "Button_20" at 954,730 size 100x68; TextOff 'Alarm Setup'
      on Click: ActivateScreen("Alarm Setup", 0)
   Button "Button_21" at 1054,730 size 110x68; TextOff 'Alarm History'
      on Click: ActivateScreen("Alarm History", 0)

Template "Template_All" 1280x800
   GraphicView "Template_Graphic view_2" at 316,3 size 194x105; Picture "mXoqcDlI_400x400"
   TextField "Template_Text field_1" at 826,19 size 97x81; Text 'bar'
   IOField "Template_I/O field_3" at 525,2 size 262x99; FormatPattern 99.9
      ProcessValue <- "ANALOG_DISPLAY.STEAM_PRESSURE"
   GraphicView "Template_Graphic view_1" at 10,6 size 125x97; Picture "euroasiatic_jaya"
   GraphicView "Template_Graphic view_3" at 139,7 size 172x96; Picture "ACTOM"
   DateTimeField "Template_Date/time field_1" at 1080,8 size 155x40
   DateTimeField "Template_Date/time field_2" at 1080,63 size 169x40
   Button "Template_Button_2" at 1058,2 size 220x52; TextOff 'Text'
      on Click: function_efd93a16("Change Date Time", 540, 220, -1, -1, 1)
   Button "Template_Button_1" at 1058,57 size 220x52; TextOff 'Text'
      on Click: function_efd93a16("Change Date Time", 540, 220, -1, -1, 1)
   Button "Template_Button_3" at 10,6 size 125x97; TextOff 'Text'
      on Click: StopRuntime(0)

Template "Template_Home" 1280x800
   GraphicView "Template_Graphic view_2" at 316,3 size 194x105; Picture "mXoqcDlI_400x400"
   GraphicView "Template_Graphic view_1" at 10,6 size 125x97; Picture "euroasiatic_jaya"
   GraphicView "Template_Graphic view_3" at 139,7 size 172x96; Picture "ACTOM"
   TextField "Template_Text field_1" at 826,19 size 97x81; Text 'bar'
   IOField "Template_I/O field_3" at 525,2 size 262x99; FormatPattern 99.9
      ProcessValue <- "ANALOG_DISPLAY.STEAM_PRESSURE"
   DateTimeField "Template_Date/time field_1" at 1082,7 size 155x40
   Button "Template_Button_2" at 1058,2 size 220x52; TextOff 'Text'
      on Click: function_efd93a16("Change Date Time", 540, 220, -1, -1, 1)
   DateTimeField "Template_Date/time field_2" at 1082,62 size 169x40
   Button "Template_Button_1" at 1058,57 size 220x52; TextOff 'Text'
      on Click: function_efd93a16("Change Date Time", 540, 220, -1, -1, 1)
   Button "Template_Button_3" at 10,6 size 125x97; TextOff 'Text'
      on Click: StopRuntime(0)

PopupScreen "Automatic Blowdown" 240x240
   Button "Button_1" at 201,9 size 34x26; TextOff 'X'
      on Click: ActivateScreen("Home Screen", 0)
   TextField "Text field_1" at 25,11 size 178x20; Text 'AUTOMATIC BLOWDOWN'
   TextField "Text field_2" at 12,122 size 73x22; Text 'OFF TIME'
   TextField "Text field_3" at 10,149 size 78x22; Text 'OFF PULSE'
   TextField "Text field_14" at 13,175 size 72x22; Text 'ON PULSE'
   TextField "Text field_15" at 16,202 size 65x22; Text 'PERIODE'
   TextField "Text field_16" at 171,120 size 28x22; Text 'min'
   TextField "Text field_17" at 171,147 size 27x22; Text 'sec'
   TextField "Text field_18" at 171,173 size 27x22; Text 'sec'
   TextField "Text field_19" at 165,203 size 40x22; Text 'times'
   Switch "Switch_3" at 75,78 size 89x32; TextOn 'ON'; CaptionText 'Switch'; TextOff 'OFF'
      ProcessValue <- "PB_BLOWDOWN"
      Appearance <- "PB_BLOWDOWN"
   IOField "I/O field_1" at 92,120 size 53x26; FormatPattern 999
      ProcessValue <- "DATA_PARAMETER.OFF_TIME_BLOWDOWN"
   IOField "I/O field_2" at 92,147 size 53x26; FormatPattern 999
      ProcessValue <- "DATA_PARAMETER.OFF_PULSE_BLOWDOWN"
   IOField "I/O field_3" at 92,174 size 53x26; FormatPattern 999
      ProcessValue <- "DATA_PARAMETER.ON_PULSE_BLOWDOWN"
   IOField "I/O field_4" at 92,201 size 53x26; FormatPattern 999
      ProcessValue <- "DATA_PARAMETER.PERIODE"
   Switch "Switch_1" at 75,44 size 89x32; TextOn 'AUTO'; CaptionText 'Switch'; TextOff 'HAND'
      ProcessValue <- "Hand/Auto_Blowdown"
      Appearance <- "Hand/Auto_Blowdown"

PopupScreen "Change Date Time" 402x252
   TextField "Text field_1" at 29,16 size 285x25; Text 'Change system date and time'
   TextField "Text field_2" at 5,81 size 78x25; Text 'Actual :'
   TextField "Text field_3" at 5,142 size 145x25; Text 'Set date time :'
   Button "Button_1" at 344,10 size 47x36; TextOff 'X'
      on Click: function_efd93a16("Change Date Time", 0, 0, -1, -1, 1)
   Button "Button_2" at 12,195 size 374x44; TextOff 'Change'
      on Press: function_b14e0dd5("Set_DTL", 0)
      Appearance <- "Set_DTL"
   IOField "I/O field_1" at 138,136 size 248x38; FormatPattern 9999999999999999999999999999999999999999
      ProcessValue <- "Set_Date_Time"
   IOField "I/O field_2" at 138,75 size 248x38; FormatPattern 9999999999999999999999999999999999999999
      ProcessValue <- "Date_Time_Actual"

PopupScreen "BURN_BACK_OFFSET LH" 240x100
   TextField "Text field_1" at 7,57 size 88x25; Text 'OFFSET :'
   IOField "I/O field_1" at 96,53 size 96x32; FormatPattern 999.9
      ProcessValue <- "LH_BURN_BACK_OFFSET"
   TextField "Text field_2" at 17,13 size 153x25; Text 'LH BURN BACK'
   Button "Button_1" at 183,9 size 46x36; TextOff 'X'
      on Click: function_efd93a16("BURN_BACK_OFFSET LH", 0, 0, -1, -1, 1)

PopupScreen "BURN_BACK_OFFSET RH" 240x100
   TextField "Text field_1" at 7,57 size 88x25; Text 'OFFSET :'
   IOField "I/O field_1" at 96,53 size 96x32; FormatPattern 999.9
      ProcessValue <- "RH_BURN_BACK_OFFSET"
   TextField "Text field_2" at 17,13 size 155x25; Text 'RH BURN BACK'
   Button "Button_1" at 183,9 size 46x36; TextOff 'X'
      on Click: function_efd93a16("BURN_BACK_OFFSET RH", 0, 0, -1, -1, 1)

screen "AI Min Max Setting" 1280x800, template "Template_All"
   TextField "Text field_3" at 401,110 size 533x50; Text 'ANALOG MIN MAX PARAMETER'
   TextField "Text field_2" at 11,273 size 120x25; Text 'Scalling Min'
   TextField "Text field_4" at 11,307 size 124x25; Text 'Scalling Max'
   TextField "Text field_5" at 141,181 size 94x46; Text 'Pressure Steam'
   IOField "I/O field_1" at 141,269 size 96x32; FormatPattern 999999.9
      ProcessValue <- "DB_Scalling_Pressurre_Steam_Min"
   IOField "I/O field_2" at 141,303 size 96x32; FormatPattern 999999.9
      ProcessValue <- "DB_Scalling_Pressure_Steam_Max"
   TextField "Text field_1" at 281,181 size 88x46; Text 'Pressure Pump'
   IOField "I/O field_3" at 285,269 size 96x32; FormatPattern 999999.9
      ProcessValue <- "DB_Scalling_Pressure_Pump_Min"
   IOField "I/O field_4" at 285,303 size 96x32; FormatPattern 999999.9
      ProcessValue <- "DB_Scalling_Pressure_Pump_Max"
   TextField "Text field_6" at 427,181 size 88x46; Text 'Water Flowrate'
   IOField "I/O field_5" at 429,269 size 96x32; FormatPattern 999999.9
      ProcessValue <- "DB_Scalling_Water_Flowrate_Min"
   IOField "I/O field_6" at 429,303 size 96x32; FormatPattern 999999.9
      ProcessValue <- "DB_Scalling_Water_Flowrate_Max"
   TextField "Text field_7" at 573,181 size 76x46; Text 'Feed Pump 1'
   IOField "I/O field_7" at 573,269 size 96x32; FormatPattern 999999.9
      ProcessValue <- "DB_Scalling_Feed_Pump_1_Min"
   IOField "I/O field_8" at 573,303 size 96x32; FormatPattern 999999.9
      ProcessValue <- "DB_Scalling_Feed_Pump_1_Max"
   TextField "Text field_8" at 717,181 size 76x46; Text 'Feed Pump 2'
   IOField "I/O field_9" at 717,269 size 96x32; FormatPattern 999999.9
      ProcessValue <- "DB_Scalling_Feed_Pump_2_Min"
   IOField "I/O field_10" at 717,303 size 96x32; FormatPattern 999999.9
      ProcessValue <- "DB_Scalling_Feed_Pump_2_Max"
   TextField "Text field_9" at 861,181 size 39x46; Text 'ID Fan'
   IOField "I/O field_11" at 861,269 size 96x32; FormatPattern 999999.9
      ProcessValue <- "DB_Scalling_ID_Fan_Min"
   IOField "I/O field_12" at 861,303 size 96x32; FormatPattern 999999.9
      ProcessValue <- "DB_Scalling_ID_Fan_Max"
   TextField "Text field_10" at 1005,181 size 62x46; Text 'LH FD Fan'
   IOField "I/O field_13" at 1005,269 size 96x32; FormatPattern 999999.9
      ProcessValue <- "DB_Scalling_LH_FD_Fan_Min"
   IOField "I/O field_14" at 1005,303 size 96x32; FormatPattern 999999.9
      ProcessValue <- "DB_Scalling_LH_FD_Fan_Max"
   TextField "Text field_11" at 1150,181 size 64x46; Text 'RH FD Fan'
   IOField "I/O field_15" at 1150,269 size 96x32; FormatPattern 999999.9
      ProcessValue <- "DB_Scalling_RH_FD_Fan_Min"
   IOField "I/O field_16" at 1150,303 size 96x32; FormatPattern 999999.9
      ProcessValue <- "DB_Scalling_RH_FD_Fan_Max"
   TextField "Text field_12" at 141,358 size 67x46; Text 'LH Stoker'
   IOField "I/O field_17" at 141,446 size 96x32; FormatPattern 999999.9
      ProcessValue <- "DB_Scalling_LH_Stoker_Min"
   IOField "I/O field_18" at 141,480 size 96x32; FormatPattern 999999.9
      ProcessValue <- "DB_Scalling_LH_Stoker_Max"
   TextField "Text field_13" at 285,358 size 67x46; Text 'RH Stoker'
   IOField "I/O field_19" at 285,446 size 96x32; FormatPattern 999999.9
      ProcessValue <- "DB_Scalling_RH_Stoker_Min"
   IOField "I/O field_20" at 285,480 size 96x32; FormatPattern 999999.9
      ProcessValue <- "DB_Scalling_RH_Stoker_Max"
   TextField "Text field_14" at 429,358 size 61x46; Text 'NRGT Water'
   IOField "I/O field_21" at 429,446 size 96x32; FormatPattern 999999.9
      ProcessValue <- "DB_Scalling_NRGT(Water_Level)_Min"
   IOField "I/O field_22" at 429,480 size 96x32; FormatPattern 999999.9
      ProcessValue <- "DB_Scalling_NRGT(Water_Level)_Max"
   TextField "Text field_15" at 573,358 size 60x46; Text 'O2 Probe'
   IOField "I/O field_23" at 573,446 size 96x32; FormatPattern 999999.9
      ProcessValue <- "DB_Scalling_O2_Probe_Min"
   IOField "I/O field_24" at 573,480 size 96x32; FormatPattern 999999.9
      ProcessValue <- "DB_Scalling_O2_Probe_Max"
   TextField "Text field_16" at 717,358 size 62x46; Text 'Water Temp'
   IOField "I/O field_25" at 717,446 size 96x32; FormatPattern 999999.9
      ProcessValue <- "DB_Scalling_Water_Temp_Min"
   IOField "I/O field_26" at 717,480 size 96x32; FormatPattern 999999.9
      ProcessValue <- "DB_Scalling_Water_Temp_Max"
   TextField "Text field_17" at 861,358 size 56x46; Text 'Flue Temp'
   IOField "I/O field_27" at 861,446 size 96x32; FormatPattern 999999.9
      ProcessValue <- "DB_Scalling_Flue_Min"
   IOField "I/O field_28" at 861,480 size 96x32; FormatPattern 999999.9
      ProcessValue <- "DB_Scalling_Flue_Max"
   TextField "Text field_18" at 1005,358 size 76x46; Text 'LH Thermo'
   IOField "I/O field_29" at 1005,446 size 96x32; FormatPattern 999999.9
      ProcessValue <- "DB_Scalling_LH_Thermocouple_Min"
   IOField "I/O field_30" at 1005,480 size 96x32; FormatPattern 999999.9
      ProcessValue <- "DB_Scalling_LH_Thermocouple_Max"
   TextField "Text field_19" at 1150,358 size 76x46; Text 'RH Thermo'
   IOField "I/O field_31" at 1150,446 size 96x32; FormatPattern 999999.9
      ProcessValue <- "DB_Scalling_RH_Thermocouple_Min"
   IOField "I/O field_32" at 1150,480 size 96x32; FormatPattern 999999.9
      ProcessValue <- "DB_Scalling_RH_Thermocouple_Max"
   TextField "Text field_20" at 141,535 size 112x46; Text 'LH Front Undergrate'
   IOField "I/O field_33" at 141,622 size 96x32; FormatPattern 999999.9
      ProcessValue <- "DB_Scalling_LH_Front_Undergrate_Min"
   IOField "I/O field_34" at 141,656 size 96x32; FormatPattern 999999.9
      ProcessValue <- "DB_Scalling_LH_Front_Undergrate_Max"
   TextField "Text field_21" at 285,535 size 112x46; Text 'RH Front Undergrate'
   IOField "I/O field_35" at 285,622 size 96x32; FormatPattern 999999.9
      ProcessValue <- "DB_Scalling_RH_Front_Undergrate_Min"
   IOField "I/O field_36" at 285,656 size 96x32; FormatPattern 999999.9
      ProcessValue <- "DB_Scalling_RH_Front_Undergrate_Max"
   TextField "Text field_22" at 427,535 size 112x46; Text 'LH Rear Undergrate'
   IOField "I/O field_37" at 429,622 size 96x32; FormatPattern 999999.9
      ProcessValue <- "DB_Scalling_LH_Rear_Undergrate_Min"
   IOField "I/O field_38" at 429,656 size 96x32; FormatPattern 999999.9
      ProcessValue <- "DB_Scalling_LH_Rear_Undergrate_Max"
   TextField "Text field_23" at 573,535 size 112x46; Text 'RH Rear Undergrate'
   IOField "I/O field_39" at 573,622 size 96x32; FormatPattern 999999.9
      ProcessValue <- "DB_Scalling_RH_Rear_Undergrate_Min"
   IOField "I/O field_40" at 573,656 size 96x32; FormatPattern 999999.9
      ProcessValue <- "DB_Scalling_RH_Rear_Undergrate_Max"
   TextField "Text field_25" at 11,239 size 123x25; Text 'Actual Value'
   IOField "I/O field_41" at 141,235 size 96x32; FormatPattern 999999.9
      ProcessValue <- "ANALOG_DISPLAY.STEAM_PRESSURE"
   IOField "I/O field_42" at 285,235 size 96x32; FormatPattern 999999.9
      ProcessValue <- "ANALOG_DISPLAY.PUMP_PRESSURE"
   IOField "I/O field_43" at 429,235 size 96x32; FormatPattern 999999.9
      ProcessValue <- "ANALOG_DISPLAY.WATER_FLOWRATE"
   IOField "I/O field_44" at 573,235 size 96x32; FormatPattern 999999.9
      ProcessValue <- "ANALOG_DISPLAY.FP1_SPEED"
   IOField "I/O field_45" at 717,235 size 96x32; FormatPattern 999999.9
      ProcessValue <- "ANALOG_DISPLAY.FP2_SPEED"
   IOField "I/O field_46" at 861,235 size 96x32; FormatPattern 999999.9
      ProcessValue <- "ANALOG_DISPLAY.ID_SPEED"
   IOField "I/O field_47" at 1005,235 size 96x32; FormatPattern 999999.9
      ProcessValue <- "ANALOG_DISPLAY.LHFD_SPEED"
   IOField "I/O field_48" at 1150,235 size 96x32; FormatPattern 999999.9
      ProcessValue <- "ANALOG_DISPLAY.RHFD_SPEED"
   TextField "Text field_26" at 11,450 size 120x25; Text 'Scalling Min'
   TextField "Text field_27" at 11,484 size 124x25; Text 'Scalling Max'
   TextField "Text field_29" at 11,416 size 123x25; Text 'Actual Value'
   IOField "I/O field_49" at 141,412 size 96x32; FormatPattern 999999.9
      ProcessValue <- "ANALOG_DISPLAY.LHSTOKER_SPEED"
   IOField "I/O field_50" at 285,412 size 96x32; FormatPattern 999999.9
      ProcessValue <- "ANALOG_DISPLAY.RHSTOKER_SPEED"
   IOField "I/O field_51" at 429,412 size 96x32; FormatPattern 999999.9
      ProcessValue <- "ANALOG_DISPLAY.WATER_LEVEL"
   IOField "I/O field_52" at 573,412 size 96x32; FormatPattern 999999.9
      ProcessValue <- "ANALOG_DISPLAY.O2_LEVEL"
   IOField "I/O field_53" at 717,412 size 96x32; FormatPattern 999999.9
      ProcessValue <- "ANALOG_DISPLAY.WATER_TEMP"
   IOField "I/O field_54" at 861,412 size 96x32; FormatPattern 999999.9
      ProcessValue <- "ANALOG_DISPLAY.FLUE_GAS_TEMP"
   IOField "I/O field_55" at 1005,412 size 96x32; FormatPattern 999999.9
      ProcessValue <- "ANALOG_DISPLAY.LH_BURNBACK_TEMP"
   IOField "I/O field_56" at 1150,412 size 96x32; FormatPattern 999999.9
      ProcessValue <- "ANALOG_DISPLAY.RH_BURNBACK_TEMP"
   TextField "Text field_30" at 11,626 size 120x25; Text 'Scalling Min'
   TextField "Text field_31" at 11,660 size 124x25; Text 'Scalling Max'
   TextField "Text field_32" at 11,592 size 123x25; Text 'Actual Value'
   TextField "Text field_33" at 11,694 size 130x25; Text 'Analog Input'
   TextField "Text field_34" at 11,728 size 111x25; Text 'Analog Min'
   TextField "Text field_35" at 11,761 size 115x25; Text 'Analog Max'
   IOField "I/O field_57" at 141,724 size 96x32; FormatPattern 999999.9
      ProcessValue <- "DB_Scalling_Analog_LH_Front_Min"
   IOField "I/O field_58" at 141,758 size 96x32; FormatPattern 999999.9
      ProcessValue <- "DB_Scalling_Analog_LH_Front_Max"
   IOField "I/O field_59" at 285,724 size 96x32; FormatPattern 999999.9
      ProcessValue <- "DB_Scalling_Analog_RH_Front_Min"
   IOField "I/O field_60" at 285,758 size 96x32; FormatPattern 999999.9
      ProcessValue <- "DB_Scalling_Analog_RH_Front_Max"
   IOField "I/O field_61" at 429,724 size 96x32; FormatPattern 999999.9
      ProcessValue <- "DB_Scalling_Analog_LH_Rear_Min"
   IOField "I/O field_62" at 429,758 size 96x32; FormatPattern 999999.9
      ProcessValue <- "DB_Scalling_Analog_LH_Rear_Max"
   IOField "I/O field_63" at 573,724 size 96x32; FormatPattern 999999.9
      ProcessValue <- "DB_Scalling_Analog_RH_Rear_Min"
   IOField "I/O field_64" at 573,758 size 96x32; FormatPattern 999999.9
      ProcessValue <- "DB_Scalling_Analog_RH_Rear_Max"
   IOField "I/O field_65" at 141,690 size 96x32; FormatPattern 9999999
      ProcessValue <- "DB103_ANALOG_INPUT_STAT15_Poti LH Front Undgrt"
   IOField "I/O field_66" at 285,690 size 96x32; FormatPattern 9999999
      ProcessValue <- "DB103_ANALOG_INPUT_STAT16_Poti RH Front Undgrt"
   IOField "I/O field_67" at 429,690 size 96x32; FormatPattern 9999999
      ProcessValue <- "DB103_ANALOG_INPUT_STAT17_Poti LH Rear Undgrt"
   IOField "I/O field_68" at 573,690 size 96x32; FormatPattern 9999999
      ProcessValue <- "DB103_ANALOG_INPUT_STAT18_Poti RH Rear Undgrt"
   IOField "I/O field_69" at 141,588 size 96x32; FormatPattern 999999.9
      ProcessValue <- "ANALOG_DISPLAY.LH_FRONT_UND_POS"
   IOField "I/O field_70" at 285,588 size 96x32; FormatPattern 999999.9
      ProcessValue <- "ANALOG_DISPLAY.RH_FRONT_UND_POS"
   IOField "I/O field_71" at 429,588 size 96x32; FormatPattern 999999.9
      ProcessValue <- "ANALOG_DISPLAY.LH_REAR_UND_POS"
   IOField "I/O field_72" at 573,588 size 96x32; FormatPattern 999999.9
      ProcessValue <- "ANALOG_DISPLAY.RH_REAR_UND_POS"
   Button "Button_1" at 1036,735 size 208x49; TextOff 'Home'
      on Click: ActivateScreen("Home Screen", 0)
   TextField "Text field_24" at 755,540 size 95x32; Text 'INFO !!'
      Appearance <- "Clock_1s"
   TextField "Text field_28" at 718,589 size 137x22; Text 'Pressure Steam'
   TextField "Text field_36" at 718,605 size 130x22; Text 'Pressure Pump'
   TextField "Text field_37" at 718,621 size 136x22; Text 'Water Flowrate'
   TextField "Text field_38" at 718,637 size 111x22; Text 'Feed Pump 1'
   TextField "Text field_39" at 718,653 size 111x22; Text 'Feed Pump 2'
   TextField "Text field_40" at 718,669 size 60x22; Text 'ID Fan'
   TextField "Text field_41" at 718,685 size 89x22; Text 'LH FD Fan'
   TextField "Text field_42" at 718,701 size 91x22; Text 'RH FD Fan'
   TextField "Text field_43" at 718,717 size 88x22; Text 'LH Stoker'
   TextField "Text field_44" at 718,733 size 90x22; Text 'RH Stoker'
   TextField "Text field_45" at 718,749 size 159x22; Text 'NRGT Water Level'
   TextField "Text field_46" at 718,765 size 83x22; Text 'O2 Probe'
   TextField "Text field_47" at 881,589 size 91x22; Text '% IW 100'
   TextField "Text field_48" at 881,605 size 91x22; Text '% IW 102'
   TextField "Text field_49" at 881,621 size 91x22; Text '% IW 104'
   TextField "Text field_50" at 881,637 size 91x22; Text '% IW 106'
   TextField "Text field_51" at 881,653 size 91x22; Text '% IW 108'
   TextField "Text field_52" at 881,669 size 91x22; Text '% IW 110'
   TextField "Text field_53" at 881,685 size 91x22; Text '% IW 112'
   TextField "Text field_54" at 881,701 size 91x22; Text '% IW 114'
   TextField "Text field_55" at 881,717 size 91x22; Text '% IW 200'
   TextField "Text field_56" at 881,733 size 91x22; Text '% IW 202'
   TextField "Text field_57" at 881,749 size 91x22; Text '% IW 204'
   TextField "Text field_58" at 881,765 size 91x22; Text '% IW 206'
   TextField "Text field_59" at 1030,589 size 105x22; Text 'Water Temp'
   TextField "Text field_60" at 1164,589 size 91x22; Text '% IW 300'
   TextField "Text field_61" at 1030,605 size 90x22; Text 'Flue Temp'
   TextField "Text field_62" at 1164,605 size 91x22; Text '% IW 302'
   TextField "Text field_63" at 1030,621 size 94x22; Text 'LH Thermo'
   TextField "Text field_64" at 1164,621 size 91x22; Text '% IW 308'
   TextField "Text field_65" at 1030,637 size 96x22; Text 'RH Thermo'
   TextField "Text field_66" at 1164,637 size 91x22; Text '% IW 310'
   TextField "Text field_67" at 1030,653 size 114x22; Text 'LH Front Und'
   TextField "Text field_68" at 1164,653 size 91x22; Text '% IW 208'
   TextField "Text field_69" at 1030,669 size 116x22; Text 'RH Front Und'
   TextField "Text field_70" at 1164,669 size 91x22; Text '% IW 212'
   TextField "Text field_71" at 1030,685 size 109x22; Text 'LH Rear Und'
   TextField "Text field_72" at 1164,685 size 91x22; Text '% IW 304'
   TextField "Text field_73" at 1030,701 size 111x22; Text 'RH Rear Und'
   TextField "Text field_74" at 1164,701 size 91x22; Text '% IW 312'
*)